Staubli VAL3: ASCIItoNum.pgx

public program ASCIItoNum(num& x_nAsc, num& x_nNum)
begin

  //This program is used for converting the hexadecimal ASCII code to the decimal number
  if x_nAsc>=48 and x_nAsc<=57
    x_nNum=x_nAsc-48
  elseIf x_nAsc>=65 and x_nAsc<=70
    x_nNum=x_nAsc-65+10
  endIf

end
